// TIA Portal V18 export
ORGANIZATION_BLOCK "Cyclic interrupt"   // OB30, LAD, CyclicInterrupt
TITLE = 100ms cyclic interrupt
{ S7_Optimized_Access := 'TRUE' }
VERSION : 0.1
// stored: AutoNumber true, IsIECCheckEnabled false, SetENOAutomatically false
   VAR_INPUT
      Initial_Call : Bool;   // Initial call of this OB
      Event_Count : Int;   // Events discarded
   END_VAR
BEGIN

REGION Network 2
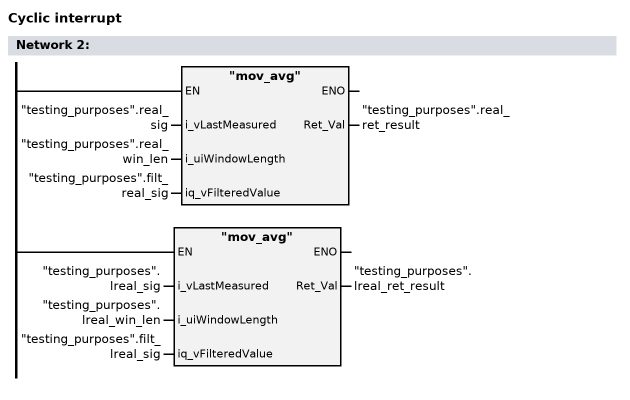
   RUNG wire#powerrail
      "mov_avg"(i_vLastMeasured := "testing_purposes".real_sig, i_uiWindowLength := "testing_purposes".real_win_len, iq_vFilteredValue := "testing_purposes".filt_real_sig, Ret_Val => "testing_purposes".real_ret_result)
   END_RUNG
   RUNG wire#powerrail
      "mov_avg"(i_vLastMeasured := "testing_purposes".lreal_sig, i_uiWindowLength := "testing_purposes".lreal_win_len, iq_vFilteredValue := "testing_purposes".filt_lreal_sig, Ret_Val => "testing_purposes".lreal_ret_result)
   END_RUNG
   // the same network as SCL:
   "testing_purposes".real_ret_result := "mov_avg"(i_vLastMeasured := "testing_purposes".real_sig,
                           i_uiWindowLength := "testing_purposes".real_win_len,
                           iq_vFilteredValue := "testing_purposes".filt_real_sig);
   "testing_purposes".lreal_ret_result := "mov_avg"(i_vLastMeasured := "testing_purposes".lreal_sig,
                           i_uiWindowLength := "testing_purposes".lreal_win_len,
                           iq_vFilteredValue := "testing_purposes".filt_lreal_sig);
END_REGION
END_ORGANIZATION_BLOCK
